Fanuc KAREL source: CA0110.KL

PROGRAM CA0110
%STACKSIZE=65535
%PRIORITY=65535
%NOLOCKGROUP
VAR
G : INTEGER
I : INTEGER
R : REAL
B : BOOLEAN
S : STRING[16]
AI : ARRAY[2] OF INTEGER
AR : ARRAY[2] OF REAL
P : XYZWPR
-- UNRESOLVED DECLARATIONS (source type spelling not recovered)
-- ST : TYPE_0x1100 (type_u16=0x1100)
-- V : TYPE_0x0013 (type_u16=0x0013)
ROUTINE F(P1 : BOOLEAN) : BOOLEAN FROM CA0110
ROUTINE F
BEGIN
RETURN(P1)
-- UNRESOLVED_PC line 22 opcodes [7F] marker_code=16
END F
BEGIN
G=0
I=1
R=2.5
B=TRUE
S='A'
AI[1]=3
AR[1]=4.5
ST.A=5
ST.B=1087373312
-- UNSAFE_SOURCE_IR line 33: CALL_RESULT F(B)
G=(G + 1)
END CA0110
